TYPE ST_CURING_STATION_SERVICE :
STRUCT
END_STRUCT
END_TYPE

(* stored: Version 1.1.0.1
   DUT ST_CURING_STATION_SERVICE: Id {f686d95d-66ee-40e4-a523-44086813a616} *)
